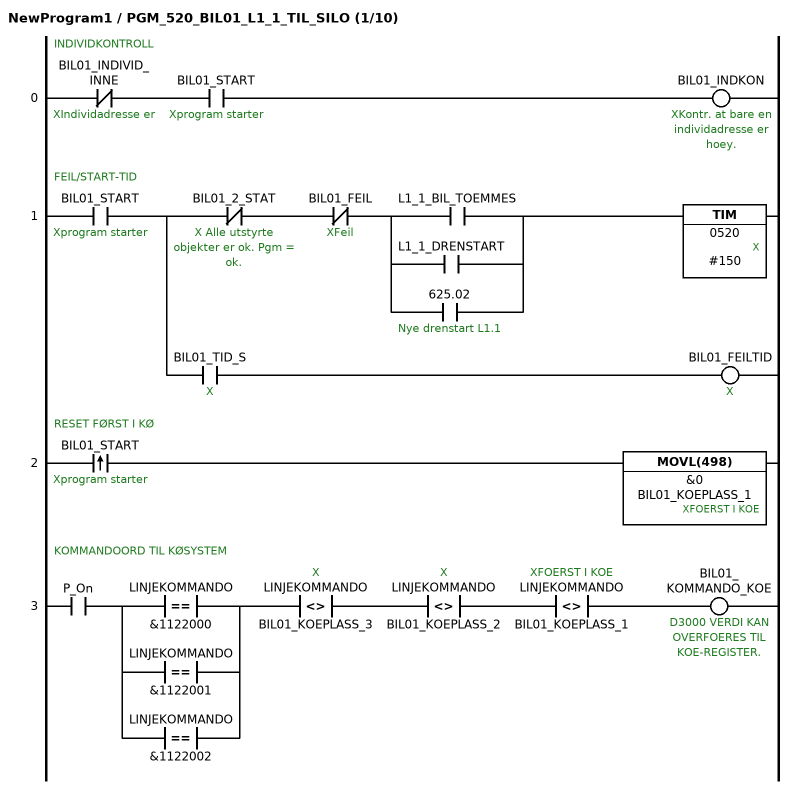
; [picture p576: NewProgram1 / PGM_520_BIL01_L1_1_TIL_SILO, rungs 0-3]
; rung 0: INDIVIDKONTROLL
LDNOT BIL01_INDIVID_INNE  ; XIndividadresse er
AND BIL01_START  ; Xprogram starter
OUT BIL01_INDKON  ; XKontr. at bare en individadresse er hoey.
; rung 1: FEIL/START-TID
LD BIL01_START  ; Xprogram starter
OUT TR0
ANDNOT BIL01_2_STAT  ; X Alle utstyrte objekter er ok. Pgm = ok.
ANDNOT BIL01_FEIL  ; XFeil
LD L1_1_BIL_TOEMMES
OR L1_1_DRENSTART
OR 625.02  ; Nye drenstart L1.1
ANDLD
TIM 0520 #150  ; X
LD TR0
AND BIL01_TID_S  ; X
OUT BIL01_FEILTID  ; X
; rung 2: RESET FØRST I KØ
@LD BIL01_START  ; Xprogram starter
MOVL(498) &0 BIL01_KOEPLASS_1  ; XFOERST I KOE
; rung 3: KOMMANDOORD TIL KØSYSTEM
LD P_On
LD=L(301) LINJEKOMMANDO &1122000
OR=L(301) LINJEKOMMANDO &1122001
OR=L(301) LINJEKOMMANDO &1122002
ANDLD
AND<>L(306) LINJEKOMMANDO BIL01_KOEPLASS_3  ; X
AND<>L(306) LINJEKOMMANDO BIL01_KOEPLASS_2  ; X
AND<>L(306) LINJEKOMMANDO BIL01_KOEPLASS_1  ; XFOERST I KOE
OUT BIL01_KOMMANDO_KOE  ; D3000 VERDI KAN OVERFOERES TIL KOE-REGISTER.

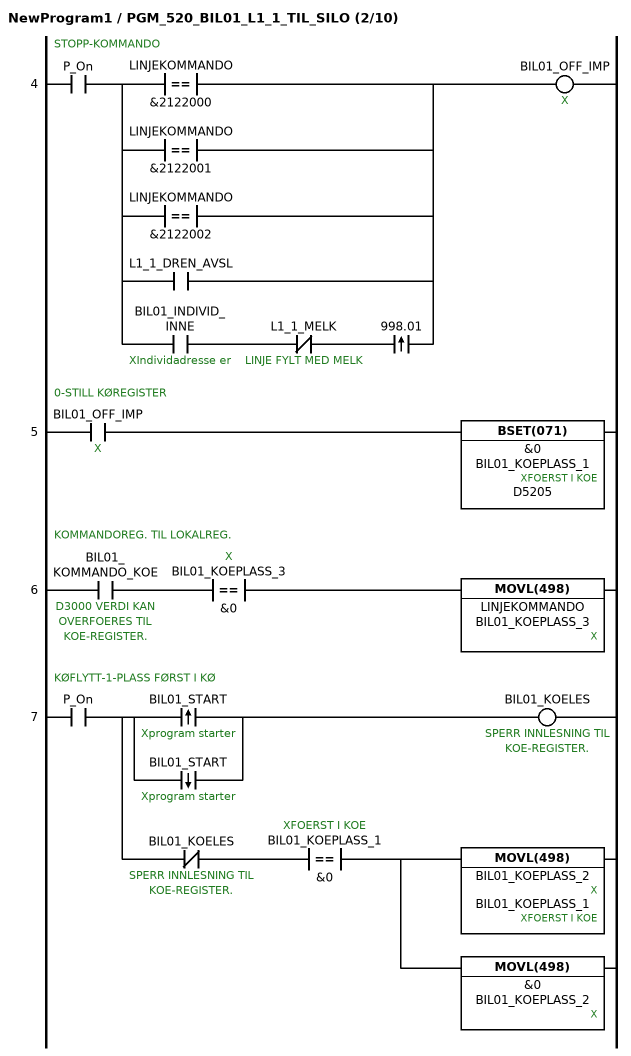
; rung 4: STOPP-KOMMANDO
LD P_On
LD=L(301) LINJEKOMMANDO &2122000
OR=L(301) LINJEKOMMANDO &2122001
OR=L(301) LINJEKOMMANDO &2122002
OR L1_1_DREN_AVSL
LD BIL01_INDIVID_INNE  ; XIndividadresse er
ANDNOT L1_1_MELK  ; LINJE FYLT MED MELK
@AND 998.01
ORLD
ANDLD
OUT BIL01_OFF_IMP  ; X
; rung 5: 0-STILL KØREGISTER
LD BIL01_OFF_IMP  ; X
BSET(071) &0 BIL01_KOEPLASS_1 D5205  ; XFOERST I KOE
; rung 6: KOMMANDOREG. TIL LOKALREG.
LD BIL01_KOMMANDO_KOE  ; D3000 VERDI KAN OVERFOERES TIL KOE-REGISTER.
AND=L(301) BIL01_KOEPLASS_3 &0  ; X
MOVL(498) LINJEKOMMANDO BIL01_KOEPLASS_3  ; X
; rung 7: KØFLYTT-1-PLASS FØRST I KØ
LD P_On
OUT TR0
@LD BIL01_START  ; Xprogram starter
%OR BIL01_START  ; Xprogram starter
ANDLD
OUT BIL01_KOELES  ; SPERR INNLESNING TIL KOE-REGISTER.
LD TR0
ANDNOT BIL01_KOELES  ; SPERR INNLESNING TIL KOE-REGISTER.
AND=L(301) BIL01_KOEPLASS_1 &0  ; XFOERST I KOE
MOVL(498) BIL01_KOEPLASS_2 BIL01_KOEPLASS_1  ; X, XFOERST I KOE
MOVL(498) &0 BIL01_KOEPLASS_2  ; X

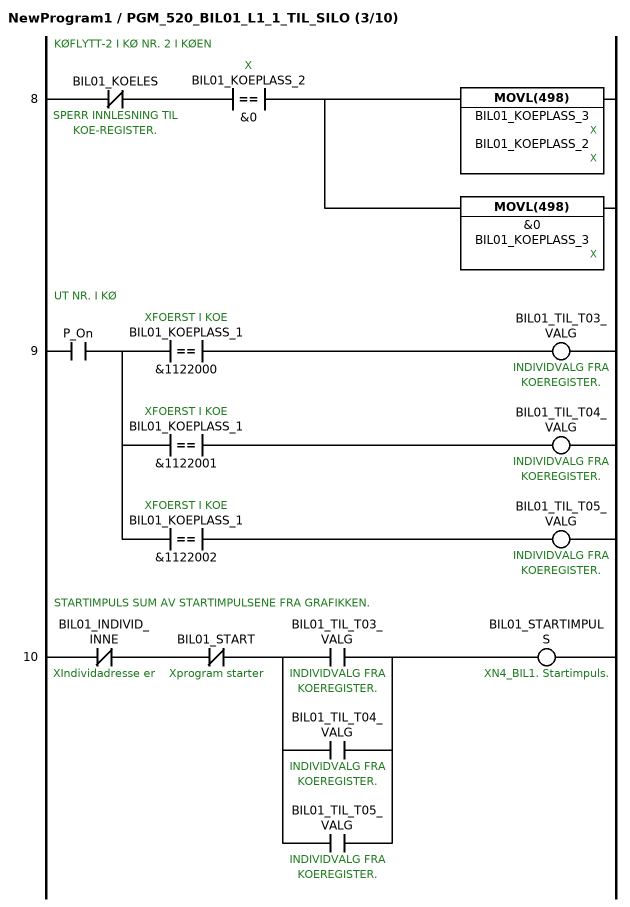
; rung 8: KØFLYTT-2 I KØ NR. 2 I KØEN
LDNOT BIL01_KOELES  ; SPERR INNLESNING TIL KOE-REGISTER.
AND=L(301) BIL01_KOEPLASS_2 &0  ; X
MOVL(498) BIL01_KOEPLASS_3 BIL01_KOEPLASS_2  ; X
MOVL(498) &0 BIL01_KOEPLASS_3  ; X
; rung 9: UT NR. I KØ
LD P_On
OUT TR0
AND=L(301) BIL01_KOEPLASS_1 &1122000  ; XFOERST I KOE
OUT BIL01_TIL_T03_VALG  ; INDIVIDVALG FRA KOEREGISTER.
LD TR0
AND=L(301) BIL01_KOEPLASS_1 &1122001  ; XFOERST I KOE
OUT BIL01_TIL_T04_VALG  ; INDIVIDVALG FRA KOEREGISTER.
LD TR0
AND=L(301) BIL01_KOEPLASS_1 &1122002  ; XFOERST I KOE
OUT BIL01_TIL_T05_VALG  ; INDIVIDVALG FRA KOEREGISTER.
; rung 10: STARTIMPULS SUM AV STARTIMPULSENE FRA GRAFIKKEN.
LDNOT BIL01_INDIVID_INNE  ; XIndividadresse er
ANDNOT BIL01_START  ; Xprogram starter
LD BIL01_TIL_T03_VALG  ; INDIVIDVALG FRA KOEREGISTER.
OR BIL01_TIL_T04_VALG  ; INDIVIDVALG FRA KOEREGISTER.
OR BIL01_TIL_T05_VALG  ; INDIVIDVALG FRA KOEREGISTER.
ANDLD
OUT BIL01_STARTIMPULS  ; XN4_BIL1. Startimpuls.

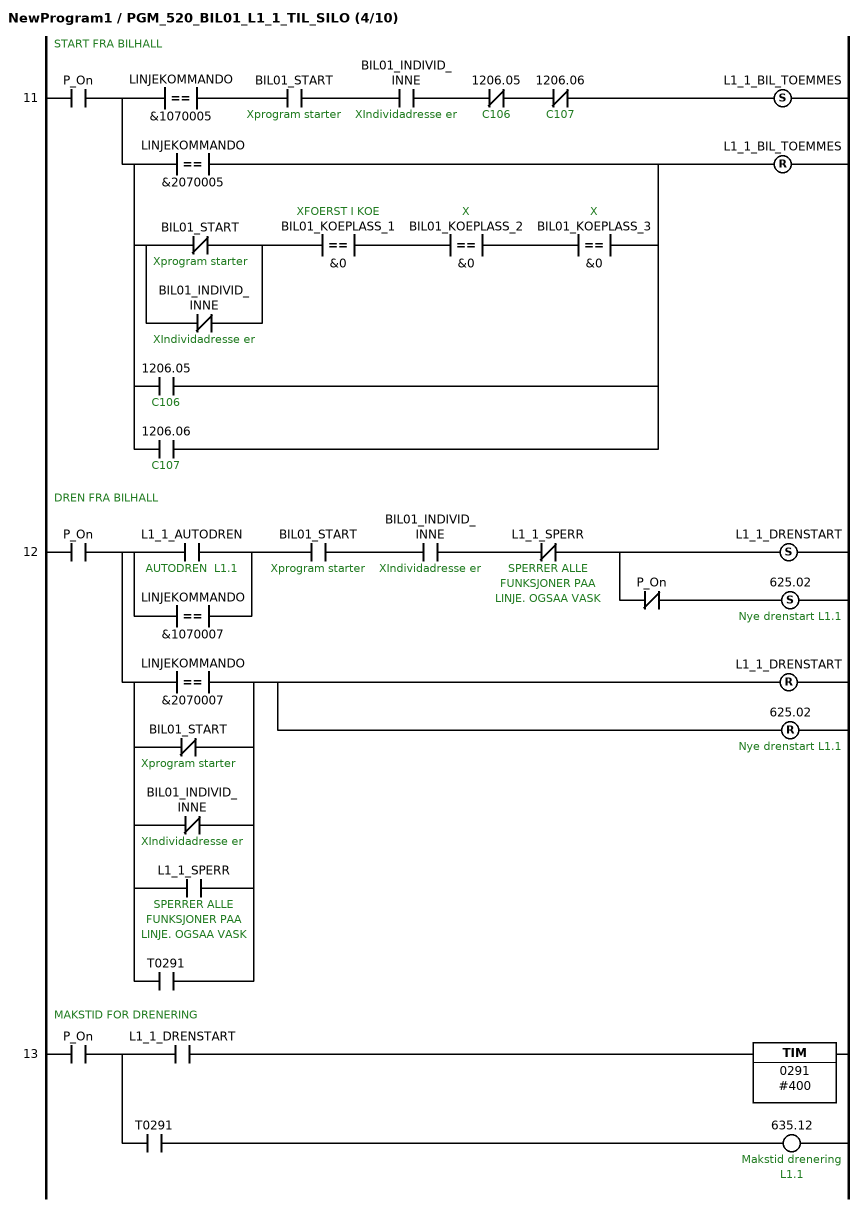
; rung 11: START FRA BILHALL
LD P_On
OUT TR0
AND=L(301) LINJEKOMMANDO &1070005
AND BIL01_START  ; Xprogram starter
AND BIL01_INDIVID_INNE  ; XIndividadresse er
ANDNOT 1206.05  ; C106
ANDNOT 1206.06  ; C107
SET L1_1_BIL_TOEMMES
LD TR0
LD=L(301) LINJEKOMMANDO &2070005
LDNOT BIL01_START  ; Xprogram starter
ORNOT BIL01_INDIVID_INNE  ; XIndividadresse er
AND=(300) BIL01_KOEPLASS_1 &0  ; XFOERST I KOE
AND=(300) BIL01_KOEPLASS_2 &0  ; X
AND=(300) BIL01_KOEPLASS_3 &0  ; X
ORLD
OR 1206.05  ; C106
OR 1206.06  ; C107
ANDLD
RSET L1_1_BIL_TOEMMES
; rung 12: DREN FRA BILHALL
LD P_On
OUT TR0
LD L1_1_AUTODREN  ; AUTODREN  L1.1
OR=L(301) LINJEKOMMANDO &1070007
ANDLD
AND BIL01_START  ; Xprogram starter
AND BIL01_INDIVID_INNE  ; XIndividadresse er
ANDNOT L1_1_SPERR  ; SPERRER ALLE FUNKSJONER PAA LINJE. OGSAA VASK
SET L1_1_DRENSTART
ANDNOT P_On
SET 625.02  ; Nye drenstart L1.1
LD TR0
LD=L(301) LINJEKOMMANDO &2070007
ORNOT BIL01_START  ; Xprogram starter
ORNOT BIL01_INDIVID_INNE  ; XIndividadresse er
OR L1_1_SPERR  ; SPERRER ALLE FUNKSJONER PAA LINJE. OGSAA VASK
OR T0291
ANDLD
RSET L1_1_DRENSTART
RSET 625.02  ; Nye drenstart L1.1
; rung 13: MAKSTID FOR DRENERING
LD P_On
OUT TR0
AND L1_1_DRENSTART
TIM 0291 #400
LD TR0
AND T0291
OUT 635.12  ; Makstid drenering L1.1

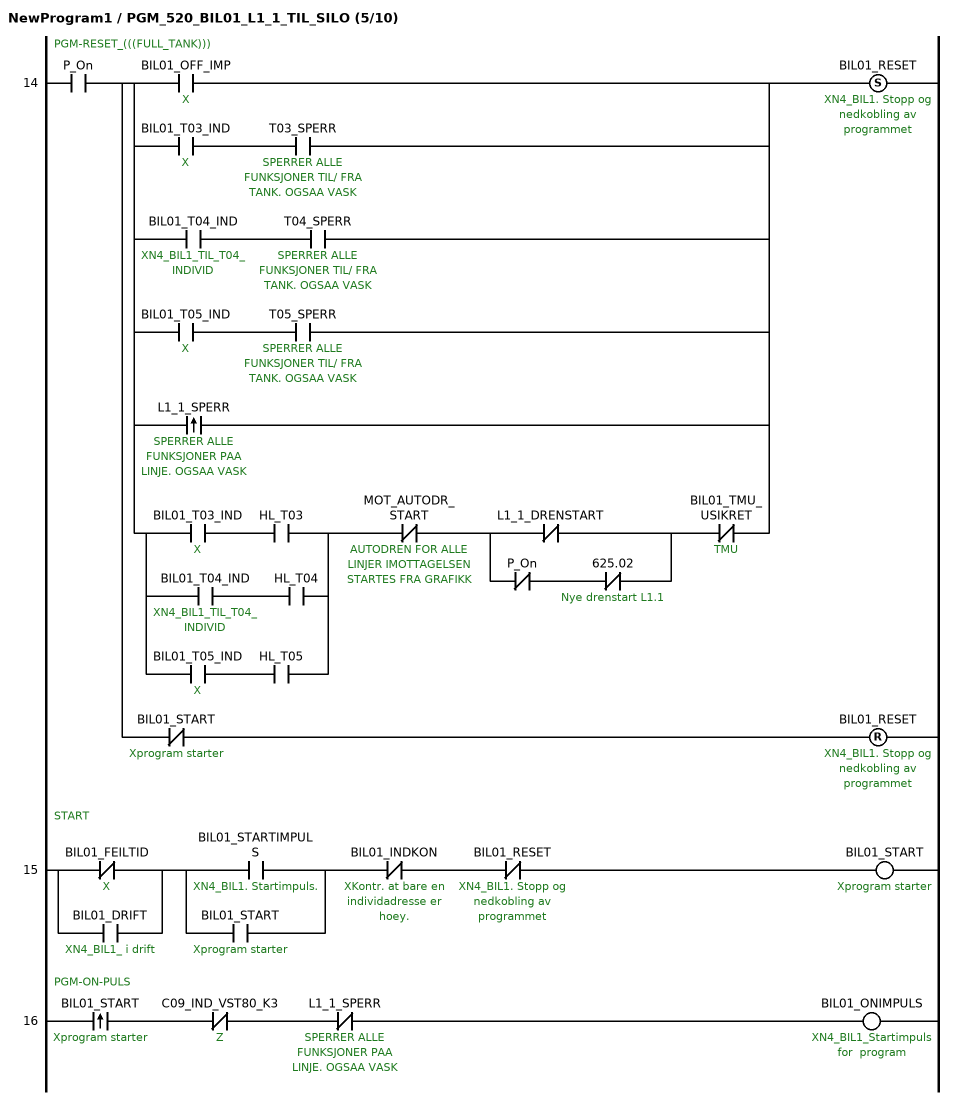
; rung 14: PGM-RESET_(((FULL_TANK)))
LD P_On
OUT TR0
LD BIL01_OFF_IMP  ; X
LD BIL01_T03_IND  ; X
AND T03_SPERR  ; SPERRER ALLE FUNKSJONER TIL/ FRA TANK. OGSAA VASK
ORLD
LD BIL01_T04_IND  ; XN4_BIL1_TIL_T04_INDIVID
AND T04_SPERR  ; SPERRER ALLE FUNKSJONER TIL/ FRA TANK. OGSAA VASK
ORLD
LD BIL01_T05_IND  ; X
AND T05_SPERR  ; SPERRER ALLE FUNKSJONER TIL/ FRA TANK. OGSAA VASK
ORLD
@OR L1_1_SPERR  ; SPERRER ALLE FUNKSJONER PAA LINJE. OGSAA VASK
LD BIL01_T03_IND  ; X
AND HL_T03
LD BIL01_T04_IND  ; XN4_BIL1_TIL_T04_INDIVID
AND HL_T04
ORLD
LD BIL01_T05_IND  ; X
AND HL_T05
ORLD
ANDNOT MOT_AUTODR_START  ; AUTODREN FOR ALLE LINJER IMOTTAGELSEN STARTES FRA GRAFIKK
LDNOT L1_1_DRENSTART
LDNOT P_On
ANDNOT 625.02  ; Nye drenstart L1.1
ORLD
ANDLD
ANDNOT BIL01_TMU_USIKRET  ; TMU
ORLD
ANDLD
SET BIL01_RESET  ; XN4_BIL1. Stopp og nedkobling av programmet
LD TR0
ANDNOT BIL01_START  ; Xprogram starter
RSET BIL01_RESET  ; XN4_BIL1. Stopp og nedkobling av programmet
; rung 15: START
LDNOT BIL01_FEILTID  ; X
OR BIL01_DRIFT  ; XN4_BIL1_ i drift
LD BIL01_STARTIMPULS  ; XN4_BIL1. Startimpuls.
OR BIL01_START  ; Xprogram starter
ANDLD
ANDNOT BIL01_INDKON  ; XKontr. at bare en individadresse er hoey.
ANDNOT BIL01_RESET  ; XN4_BIL1. Stopp og nedkobling av programmet
OUT BIL01_START  ; Xprogram starter
; rung 16: PGM-ON-PULS
@LD BIL01_START  ; Xprogram starter
ANDNOT C09_IND_VST80_K3  ; Z
ANDNOT L1_1_SPERR  ; SPERRER ALLE FUNKSJONER PAA LINJE. OGSAA VASK
OUT BIL01_ONIMPULS  ; XN4_BIL1_Startimpuls for  program

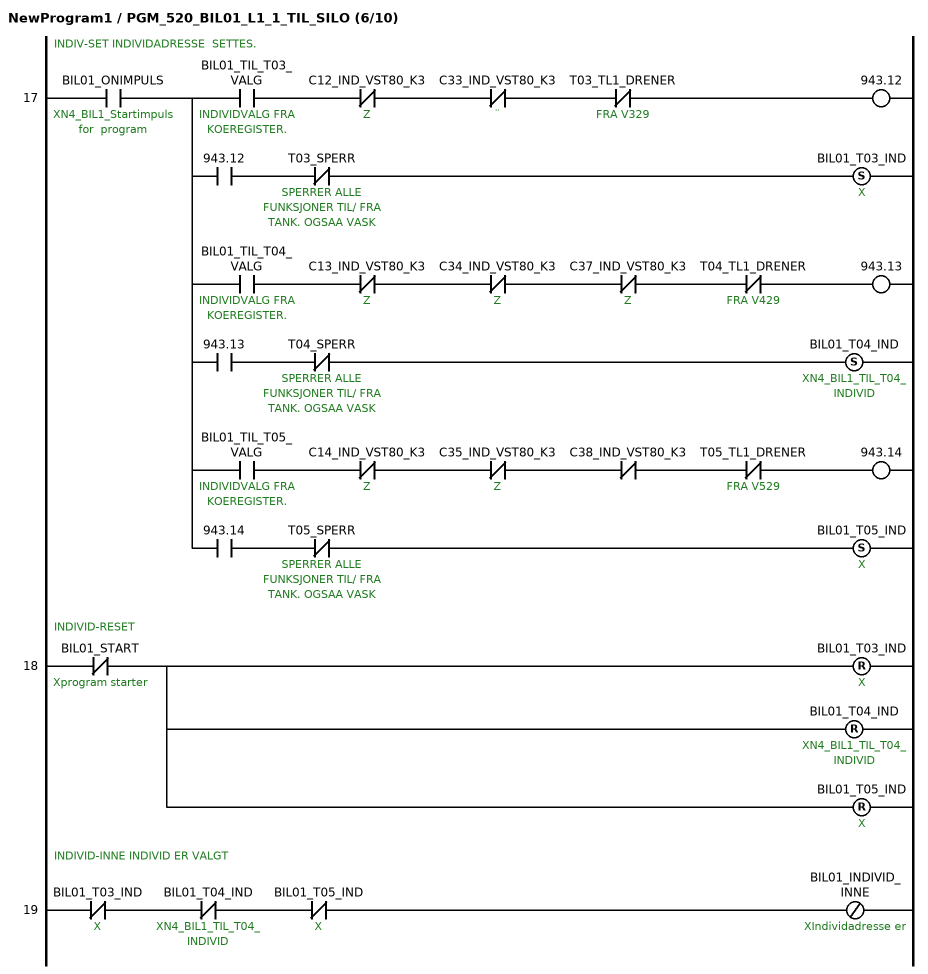
; rung 17: INDIV-SET INDIVIDADRESSE  SETTES.
LD BIL01_ONIMPULS  ; XN4_BIL1_Startimpuls for  program
OUT TR0
AND BIL01_TIL_T03_VALG  ; INDIVIDVALG FRA KOEREGISTER.
ANDNOT C12_IND_VST80_K3  ; Z
ANDNOT C33_IND_VST80_K3  ; ¨
ANDNOT T03_TL1_DRENER  ; FRA V329
OUT 943.12
LD TR0
AND 943.12
ANDNOT T03_SPERR  ; SPERRER ALLE FUNKSJONER TIL/ FRA TANK. OGSAA VASK
SET BIL01_T03_IND  ; X
LD TR0
AND BIL01_TIL_T04_VALG  ; INDIVIDVALG FRA KOEREGISTER.
ANDNOT C13_IND_VST80_K3  ; Z
ANDNOT C34_IND_VST80_K3  ; Z
ANDNOT C37_IND_VST80_K3  ; Z
ANDNOT T04_TL1_DRENER  ; FRA V429
OUT 943.13
LD TR0
AND 943.13
ANDNOT T04_SPERR  ; SPERRER ALLE FUNKSJONER TIL/ FRA TANK. OGSAA VASK
SET BIL01_T04_IND  ; XN4_BIL1_TIL_T04_INDIVID
LD TR0
AND BIL01_TIL_T05_VALG  ; INDIVIDVALG FRA KOEREGISTER.
ANDNOT C14_IND_VST80_K3  ; Z
ANDNOT C35_IND_VST80_K3  ; Z
ANDNOT C38_IND_VST80_K3
ANDNOT T05_TL1_DRENER  ; FRA V529
OUT 943.14
LD TR0
AND 943.14
ANDNOT T05_SPERR  ; SPERRER ALLE FUNKSJONER TIL/ FRA TANK. OGSAA VASK
SET BIL01_T05_IND  ; X
; rung 18: INDIVID-RESET
LDNOT BIL01_START  ; Xprogram starter
RSET BIL01_T03_IND  ; X
RSET BIL01_T04_IND  ; XN4_BIL1_TIL_T04_INDIVID
RSET BIL01_T05_IND  ; X
; rung 19: INDIVID-INNE INDIVID ER VALGT
LDNOT BIL01_T03_IND  ; X
ANDNOT BIL01_T04_IND  ; XN4_BIL1_TIL_T04_INDIVID
ANDNOT BIL01_T05_IND  ; X
OUTNOT BIL01_INDIVID_INNE  ; XIndividadresse er

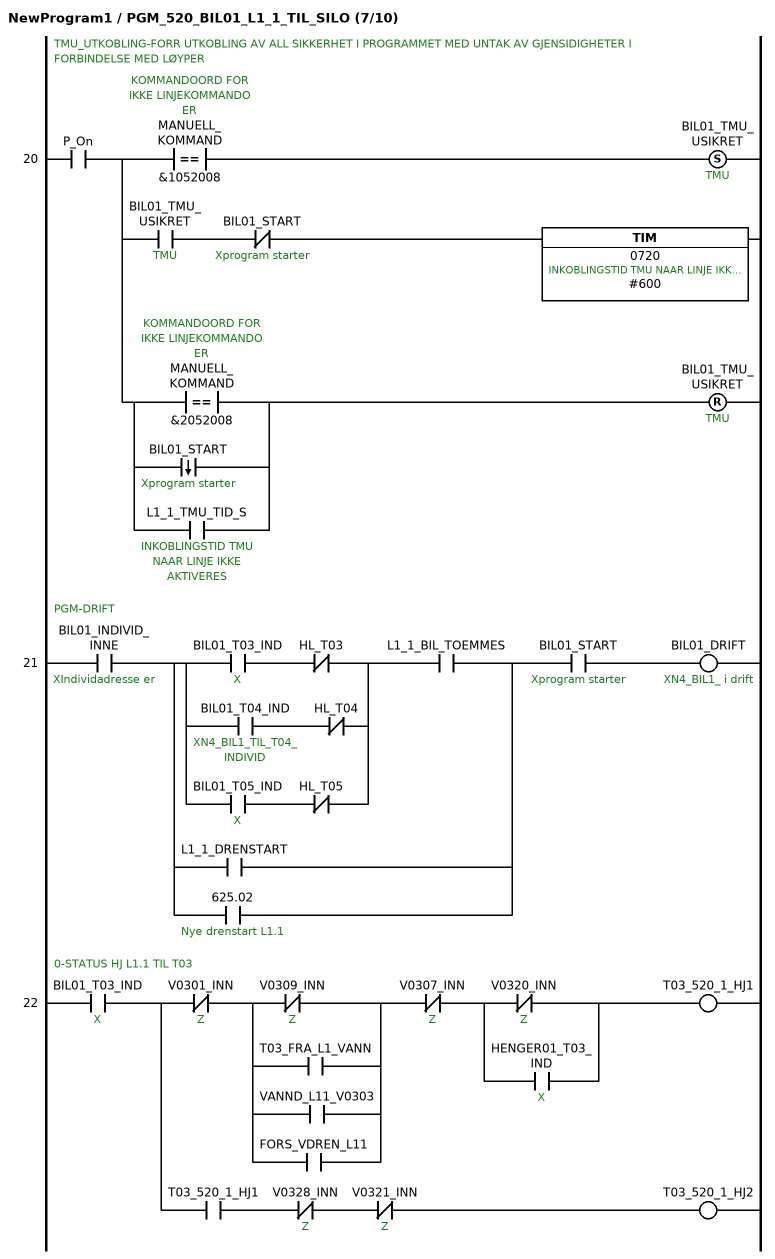
; rung 20: TMU_UTKOBLING-FORR UTKOBLING AV ALL SIKKERHET I PROGRAMMET MED UNTAK AV GJENSIDIGHETER I FORBINDELSE MED LØYPER
LD P_On
OUT TR0
AND=L(301) MANUELL_KOMMAND &1052008  ; KOMMANDOORD FOR IKKE LINJEKOMMANDOER
SET BIL01_TMU_USIKRET  ; TMU
LD TR0
AND BIL01_TMU_USIKRET  ; TMU
ANDNOT BIL01_START  ; Xprogram starter
TIM 0720 #600  ; INKOBLINGSTID TMU NAAR LINJE IKKE AKTIVERES
LD TR0
LD=L(301) MANUELL_KOMMAND &2052008  ; KOMMANDOORD FOR IKKE LINJEKOMMANDOER
%OR BIL01_START  ; Xprogram starter
OR L1_1_TMU_TID_S  ; INKOBLINGSTID TMU NAAR LINJE IKKE AKTIVERES
ANDLD
RSET BIL01_TMU_USIKRET  ; TMU
; rung 21: PGM-DRIFT
LD BIL01_INDIVID_INNE  ; XIndividadresse er
LD BIL01_T03_IND  ; X
ANDNOT HL_T03
LD BIL01_T04_IND  ; XN4_BIL1_TIL_T04_INDIVID
ANDNOT HL_T04
ORLD
LD BIL01_T05_IND  ; X
ANDNOT HL_T05
ORLD
AND L1_1_BIL_TOEMMES
OR L1_1_DRENSTART
OR 625.02  ; Nye drenstart L1.1
ANDLD
AND BIL01_START  ; Xprogram starter
OUT BIL01_DRIFT  ; XN4_BIL1_ i drift
; rung 22: 0-STATUS HJ L1.1 TIL T03
LD BIL01_T03_IND  ; X
OUT TR0
ANDNOT V0301_INN  ; Z
LDNOT V0309_INN  ; Z
OR T03_FRA_L1_VANN
OR VANND_L11_V0303
OR FORS_VDREN_L11
ANDLD
ANDNOT V0307_INN  ; Z
LDNOT V0320_INN  ; Z
OR HENGER01_T03_IND  ; X
ANDLD
OUT T03_520_1_HJ1
LD TR0
AND T03_520_1_HJ1
ANDNOT V0328_INN  ; Z
ANDNOT V0321_INN  ; Z
OUT T03_520_1_HJ2

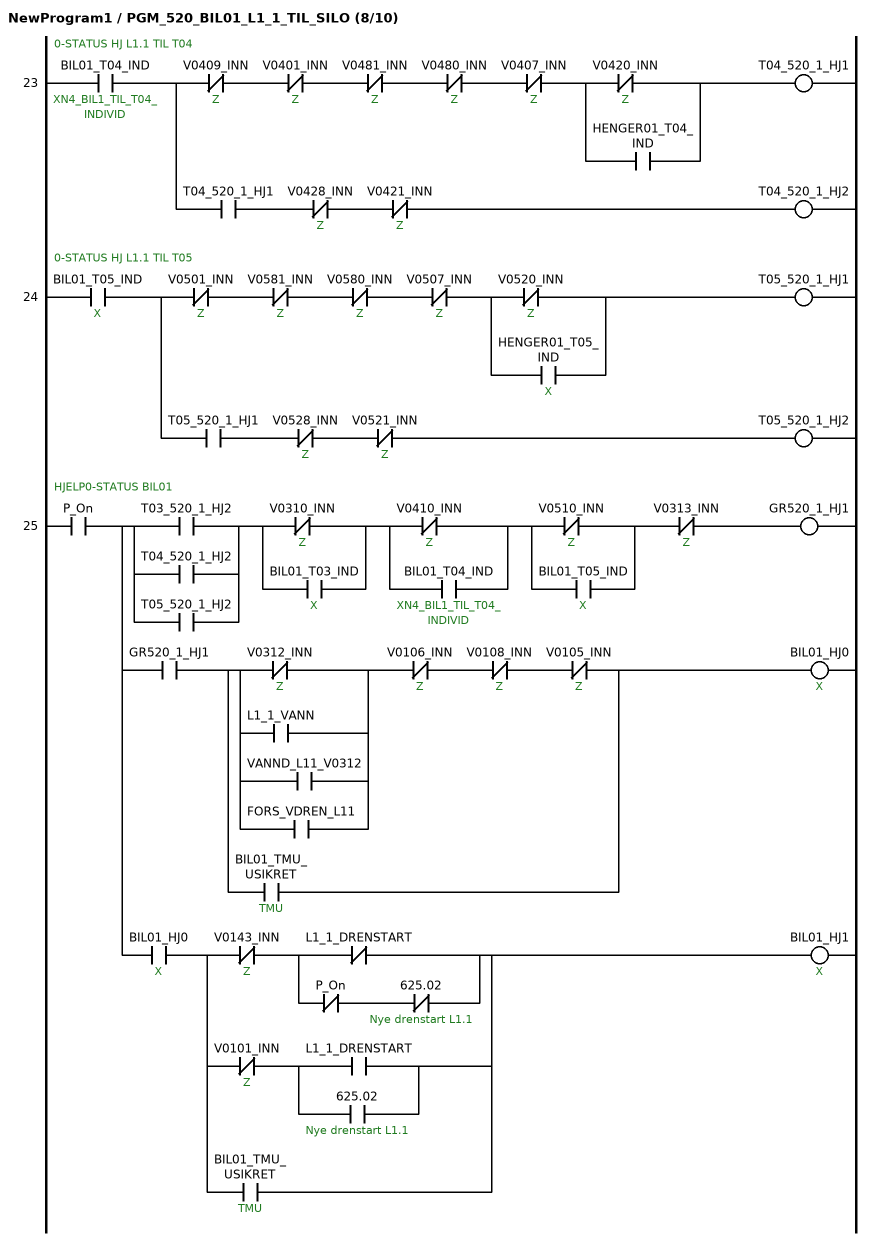
; rung 23: 0-STATUS HJ L1.1 TIL T04
LD BIL01_T04_IND  ; XN4_BIL1_TIL_T04_INDIVID
OUT TR0
ANDNOT V0409_INN  ; Z
ANDNOT V0401_INN  ; Z
ANDNOT V0481_INN  ; Z
ANDNOT V0480_INN  ; Z
ANDNOT V0407_INN  ; Z
LDNOT V0420_INN  ; Z
OR HENGER01_T04_IND
ANDLD
OUT T04_520_1_HJ1
LD TR0
AND T04_520_1_HJ1
ANDNOT V0428_INN  ; Z
ANDNOT V0421_INN  ; Z
OUT T04_520_1_HJ2
; rung 24: 0-STATUS HJ L1.1 TIL T05
LD BIL01_T05_IND  ; X
OUT TR0
ANDNOT V0501_INN  ; Z
ANDNOT V0581_INN  ; Z
ANDNOT V0580_INN  ; Z
ANDNOT V0507_INN  ; Z
LDNOT V0520_INN  ; Z
OR HENGER01_T05_IND  ; X
ANDLD
OUT T05_520_1_HJ1
LD TR0
AND T05_520_1_HJ1
ANDNOT V0528_INN  ; Z
ANDNOT V0521_INN  ; Z
OUT T05_520_1_HJ2
; rung 25: HJELP0-STATUS BIL01
LD P_On
OUT TR0
LD T03_520_1_HJ2
OR T04_520_1_HJ2
OR T05_520_1_HJ2
ANDLD
LDNOT V0310_INN  ; Z
OR BIL01_T03_IND  ; X
ANDLD
LDNOT V0410_INN  ; Z
OR BIL01_T04_IND  ; XN4_BIL1_TIL_T04_INDIVID
ANDLD
LDNOT V0510_INN  ; Z
OR BIL01_T05_IND  ; X
ANDLD
ANDNOT V0313_INN  ; Z
OUT GR520_1_HJ1
LD TR0
AND GR520_1_HJ1
LDNOT V0312_INN  ; Z
OR L1_1_VANN
OR VANND_L11_V0312
OR FORS_VDREN_L11
ANDNOT V0106_INN  ; Z
ANDNOT V0108_INN  ; Z
ANDNOT V0105_INN  ; Z
OR BIL01_TMU_USIKRET  ; TMU
ANDLD
OUT BIL01_HJ0  ; X
LD TR0
AND BIL01_HJ0  ; X
LDNOT V0143_INN  ; Z
LDNOT L1_1_DRENSTART
LDNOT P_On
ANDNOT 625.02  ; Nye drenstart L1.1
ORLD
ANDLD
LDNOT V0101_INN  ; Z
LD L1_1_DRENSTART
OR 625.02  ; Nye drenstart L1.1
ANDLD
ORLD
OR BIL01_TMU_USIKRET  ; TMU
ANDLD
OUT BIL01_HJ1  ; X

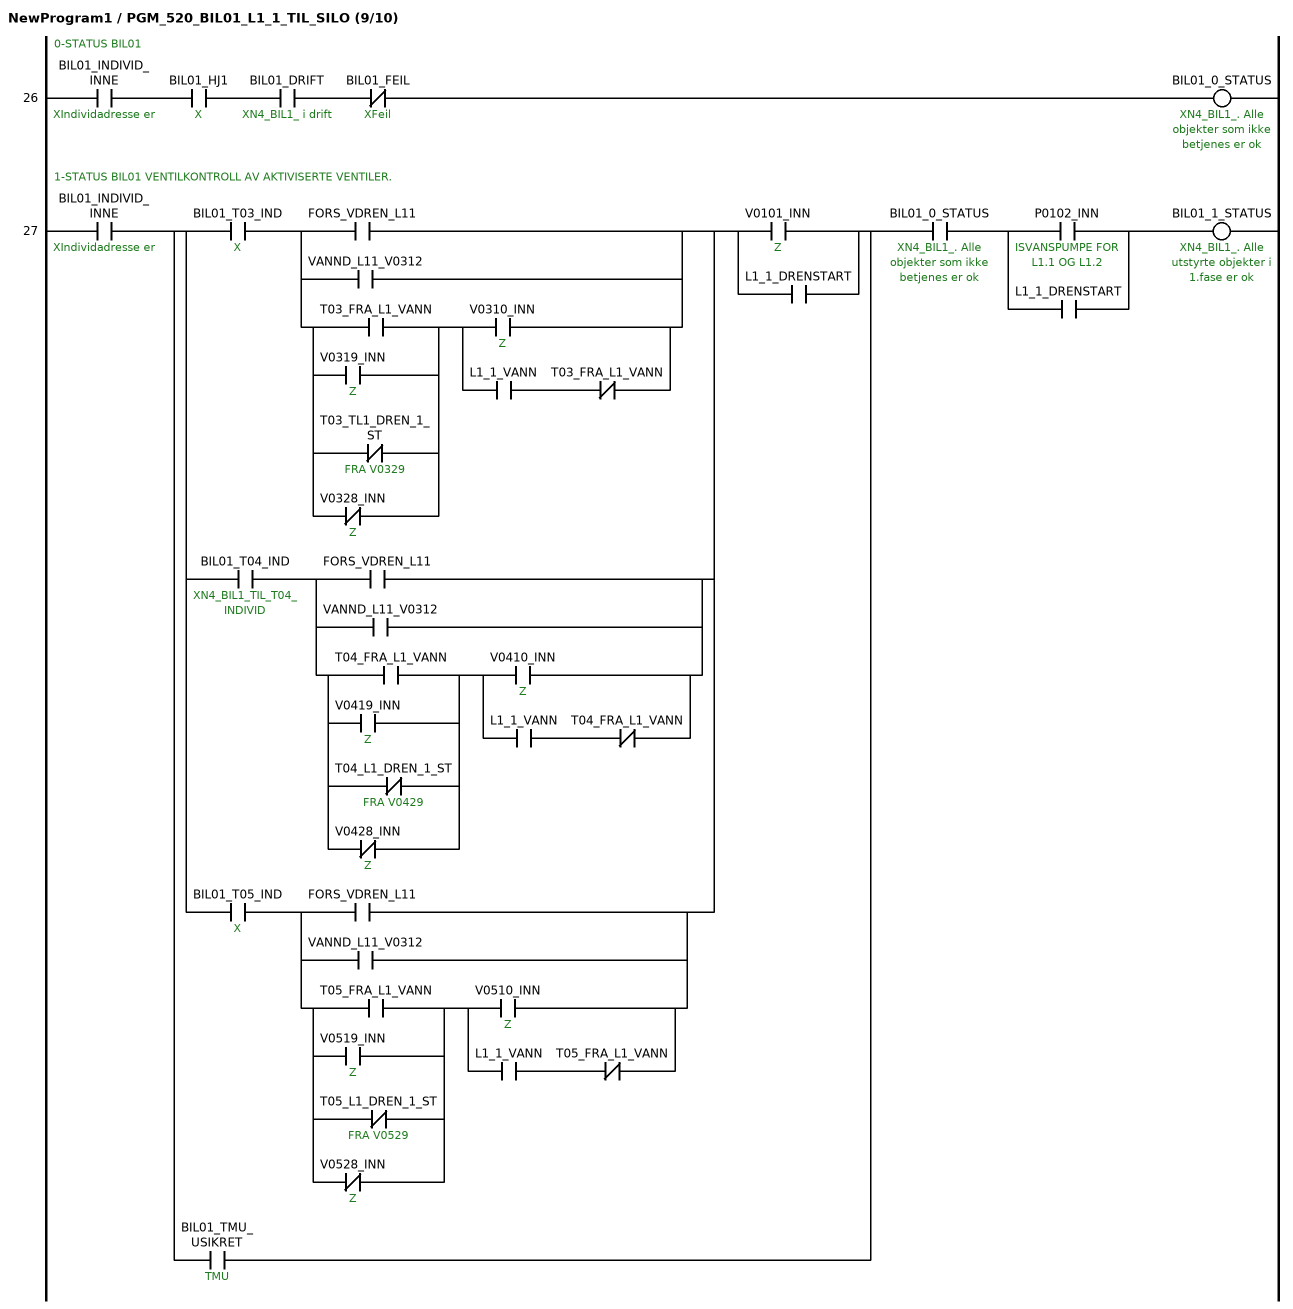
; rung 26: 0-STATUS BIL01
LD BIL01_INDIVID_INNE  ; XIndividadresse er
AND BIL01_HJ1  ; X
AND BIL01_DRIFT  ; XN4_BIL1_ i drift
ANDNOT BIL01_FEIL  ; XFeil
OUT BIL01_0_STATUS  ; XN4_BIL1_. Alle objekter som ikke betjenes er ok
; rung 27: 1-STATUS BIL01 VENTILKONTROLL AV AKTIVISERTE VENTILER.
LD BIL01_INDIVID_INNE  ; XIndividadresse er
LD BIL01_T03_IND  ; X
LD FORS_VDREN_L11
OR VANND_L11_V0312
LD T03_FRA_L1_VANN
OR V0319_INN  ; Z
ORNOT T03_TL1_DREN_1_ST  ; FRA V0329
ORNOT V0328_INN  ; Z
LD V0310_INN  ; Z
LD L1_1_VANN
ANDNOT T03_FRA_L1_VANN
ORLD
ANDLD
ORLD
ANDLD
LD BIL01_T04_IND  ; XN4_BIL1_TIL_T04_INDIVID
LD FORS_VDREN_L11
OR VANND_L11_V0312
LD T04_FRA_L1_VANN
OR V0419_INN  ; Z
ORNOT T04_L1_DREN_1_ST  ; FRA V0429
ORNOT V0428_INN  ; Z
LD V0410_INN  ; Z
LD L1_1_VANN
ANDNOT T04_FRA_L1_VANN
ORLD
ANDLD
ORLD
ANDLD
ORLD
LD BIL01_T05_IND  ; X
LD FORS_VDREN_L11
OR VANND_L11_V0312
LD T05_FRA_L1_VANN
OR V0519_INN  ; Z
ORNOT T05_L1_DREN_1_ST  ; FRA V0529
ORNOT V0528_INN  ; Z
LD V0510_INN  ; Z
LD L1_1_VANN
ANDNOT T05_FRA_L1_VANN
ORLD
ANDLD
ORLD
ANDLD
ORLD
LD V0101_INN  ; Z
OR L1_1_DRENSTART
ANDLD
OR BIL01_TMU_USIKRET  ; TMU
ANDLD
AND BIL01_0_STATUS  ; XN4_BIL1_. Alle objekter som ikke betjenes er ok
LD P0102_INN  ; ISVANSPUMPE FOR L1.1 OG L1.2
OR L1_1_DRENSTART
ANDLD
OUT BIL01_1_STATUS  ; XN4_BIL1_. Alle utstyrte objekter i 1.fase er ok

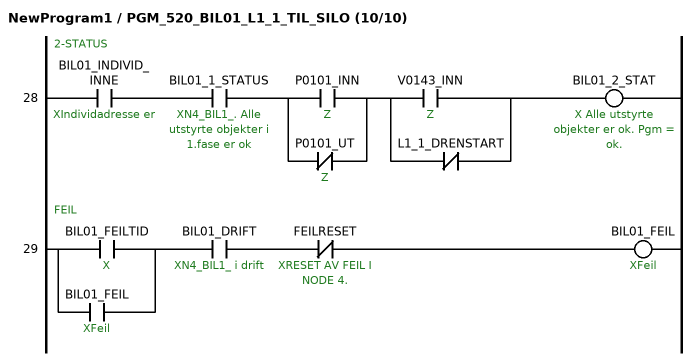
; rung 28: 2-STATUS
LD BIL01_INDIVID_INNE  ; XIndividadresse er
AND BIL01_1_STATUS  ; XN4_BIL1_. Alle utstyrte objekter i 1.fase er ok
LD P0101_INN  ; Z
ORNOT P0101_UT  ; Z
ANDLD
LD V0143_INN  ; Z
ORNOT L1_1_DRENSTART
ANDLD
OUT BIL01_2_STAT  ; X Alle utstyrte objekter er ok. Pgm = ok.
; rung 29: FEIL
LD BIL01_FEILTID  ; X
OR BIL01_FEIL  ; XFeil
AND BIL01_DRIFT  ; XN4_BIL1_ i drift
ANDNOT FEILRESET  ; XRESET AV FEIL I NODE 4.
OUT BIL01_FEIL  ; XFeil
; rung 30: Ingen_kommentar_funnet

### Section V0104_P0101

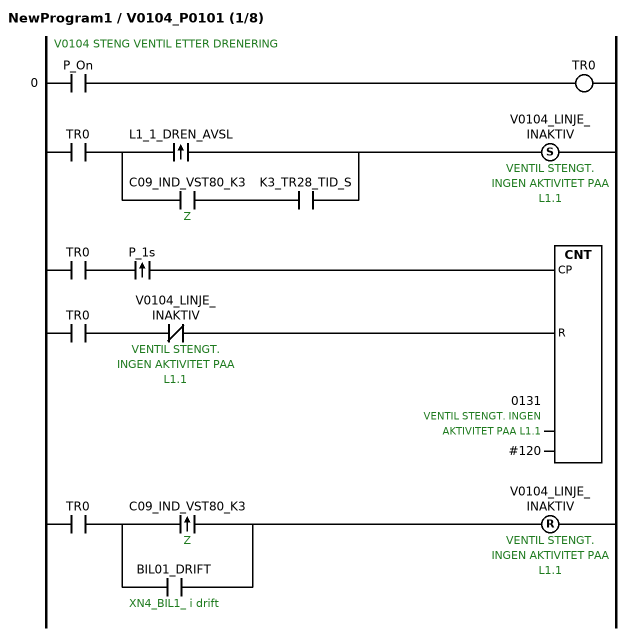
; rung 0: V0104 STENG VENTIL ETTER DRENERING
LD P_On
OUT TR0
@LD L1_1_DREN_AVSL
LD C09_IND_VST80_K3  ; Z
AND K3_TR28_TID_S
ORLD
ANDLD
SET V0104_LINJE_INAKTIV  ; VENTIL STENGT. INGEN AKTIVITET PAA L1.1
LD TR0
@AND P_1s
LD TR0
ANDNOT V0104_LINJE_INAKTIV  ; VENTIL STENGT. INGEN AKTIVITET PAA L1.1
CNT 0131 #120  ; VENTIL STENGT. INGEN AKTIVITET PAA L1.1
LD TR0
@LD C09_IND_VST80_K3  ; Z
OR BIL01_DRIFT  ; XN4_BIL1_ i drift
ANDLD
RSET V0104_LINJE_INAKTIV  ; VENTIL STENGT. INGEN AKTIVITET PAA L1.1

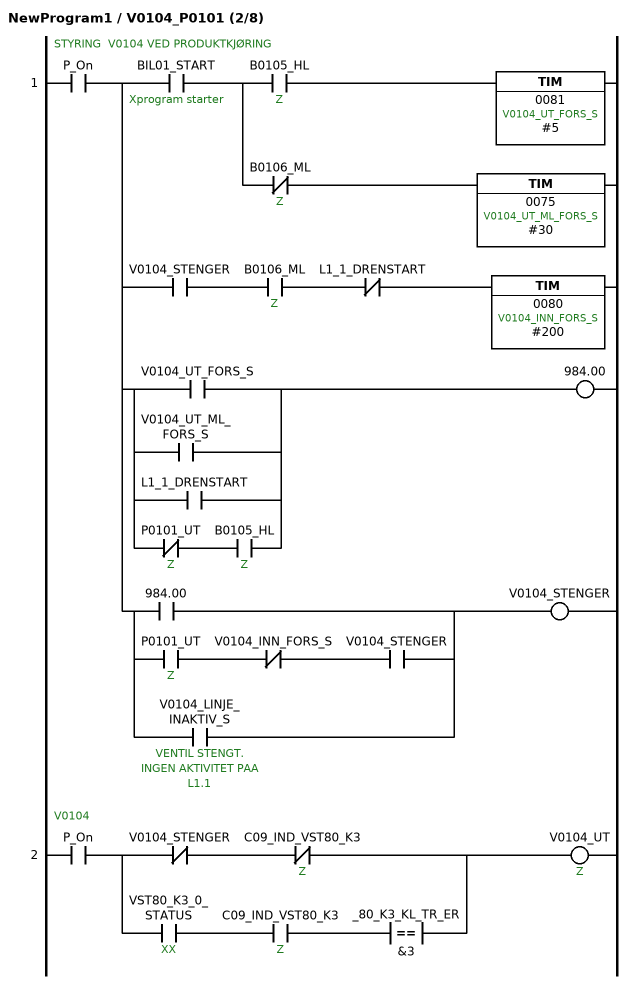
; rung 1: STYRING  V0104 VED PRODUKTKJØRING
LD P_On
OUT TR0
AND BIL01_START  ; Xprogram starter
OUT TR1
AND B0105_HL  ; Z
TIM 0081 #5  ; V0104_UT_FORS_S
LD TR1
ANDNOT B0106_ML  ; Z
TIM 0075 #30  ; V0104_UT_ML_FORS_S
LD TR0
AND V0104_STENGER
AND B0106_ML  ; Z
ANDNOT L1_1_DRENSTART
TIM 0080 #200  ; V0104_INN_FORS_S
LD TR0
LD V0104_UT_FORS_S
OR V0104_UT_ML_FORS_S
OR L1_1_DRENSTART
LDNOT P0101_UT  ; Z
AND B0105_HL  ; Z
ORLD
ANDLD
OUT 984.00
LD TR0
LD 984.00
LD P0101_UT  ; Z
ANDNOT V0104_INN_FORS_S
AND V0104_STENGER
ORLD
OR V0104_LINJE_INAKTIV_S  ; VENTIL STENGT. INGEN AKTIVITET PAA L1.1
ANDLD
OUT V0104_STENGER
; rung 2: V0104
LD P_On
LDNOT V0104_STENGER
ANDNOT C09_IND_VST80_K3  ; Z
LD VST80_K3_0_STATUS  ; XX
AND C09_IND_VST80_K3  ; Z
AND=(300) _80_K3_KL_TR_ER &3
ORLD
ANDLD
OUT V0104_UT  ; Z

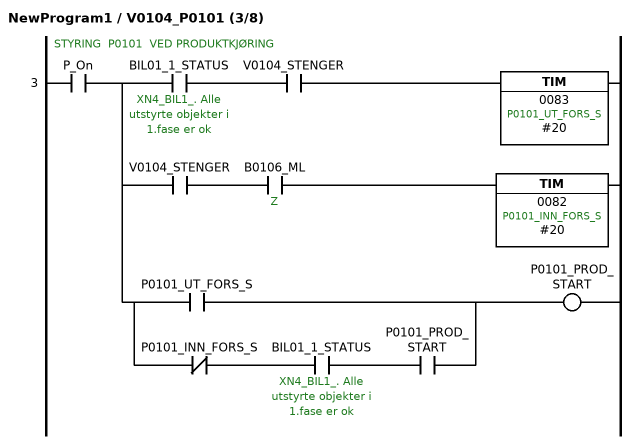
; rung 3: STYRING  P0101  VED PRODUKTKJØRING
LD P_On
OUT TR0
AND BIL01_1_STATUS  ; XN4_BIL1_. Alle utstyrte objekter i 1.fase er ok
AND V0104_STENGER
TIM 0083 #20  ; P0101_UT_FORS_S
LD TR0
AND V0104_STENGER
AND B0106_ML  ; Z
TIM 0082 #20  ; P0101_INN_FORS_S
LD TR0
LD P0101_UT_FORS_S
LDNOT P0101_INN_FORS_S
AND BIL01_1_STATUS  ; XN4_BIL1_. Alle utstyrte objekter i 1.fase er ok
AND P0101_PROD_START
ORLD
ANDLD
OUT P0101_PROD_START

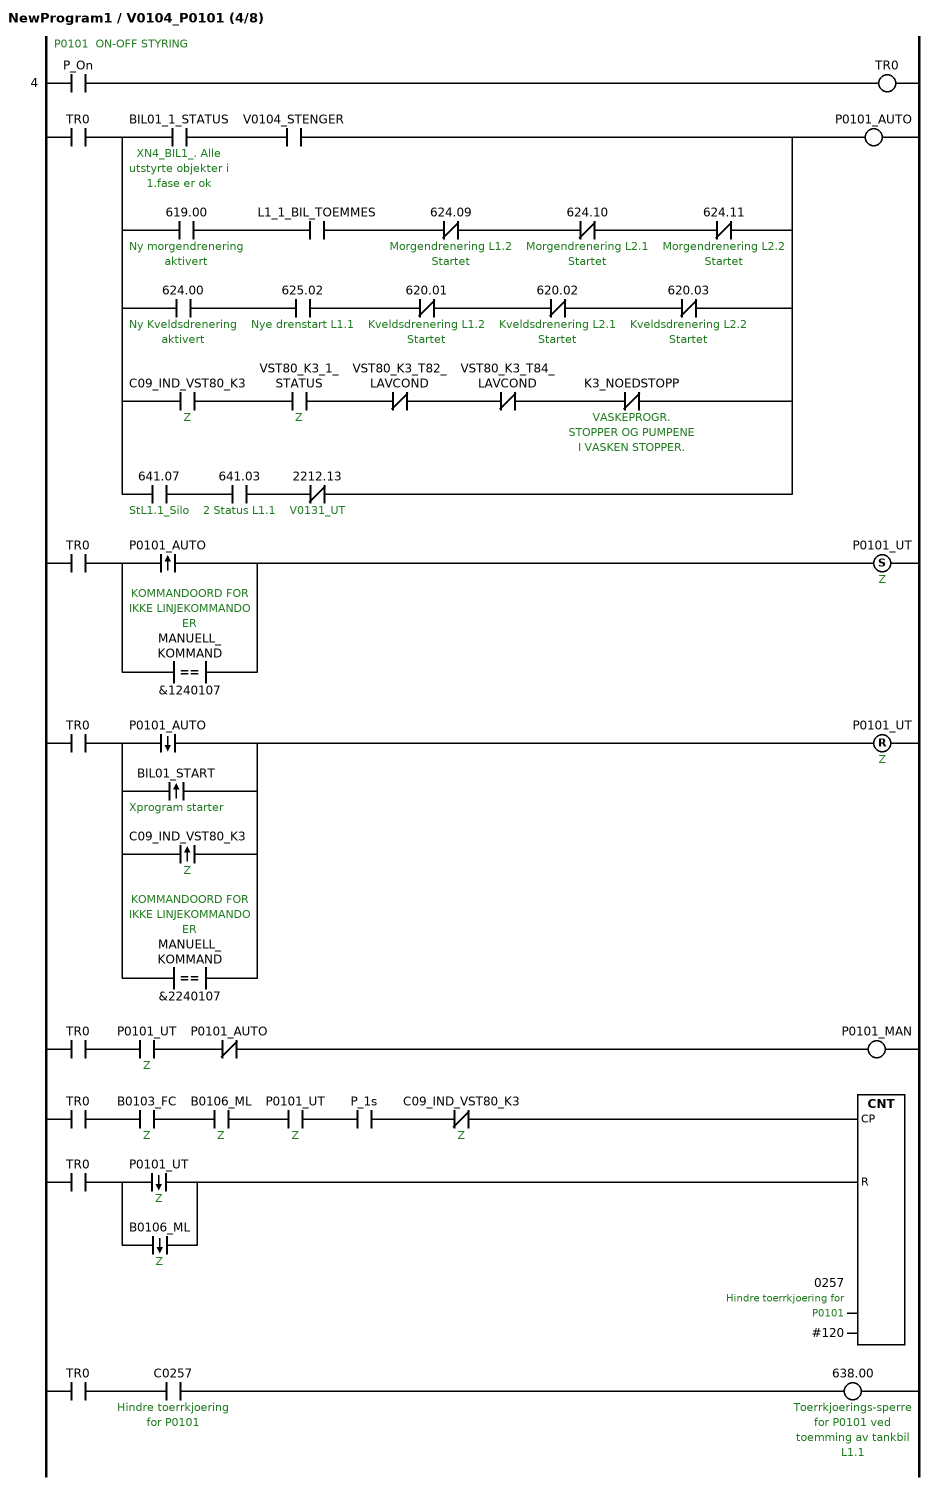
; rung 4: P0101  ON-OFF STYRING
LD P_On
OUT TR0
LD BIL01_1_STATUS  ; XN4_BIL1_. Alle utstyrte objekter i 1.fase er ok
AND V0104_STENGER
LD 619.00  ; Ny morgendrenering aktivert
AND L1_1_BIL_TOEMMES
ANDNOT 624.09  ; Morgendrenering L1.2 Startet
ANDNOT 624.10  ; Morgendrenering L2.1 Startet
ANDNOT 624.11  ; Morgendrenering L2.2 Startet
ORLD
LD 624.00  ; Ny Kveldsdrenering aktivert
AND 625.02  ; Nye drenstart L1.1
ANDNOT 620.01  ; Kveldsdrenering L1.2 Startet
ANDNOT 620.02  ; Kveldsdrenering L2.1 Startet
ANDNOT 620.03  ; Kveldsdrenering L2.2 Startet
ORLD
LD C09_IND_VST80_K3  ; Z
AND VST80_K3_1_STATUS  ; Z
ANDNOT VST80_K3_T82_LAVCOND
ANDNOT VST80_K3_T84_LAVCOND
ANDNOT K3_NOEDSTOPP  ; VASKEPROGR. STOPPER OG PUMPENE I VASKEN STOPPER.
ORLD
LD 641.07  ; StL1.1_Silo
AND 641.03  ; 2 Status L1.1
ANDNOT 2212.13  ; V0131_UT
ORLD
ANDLD
OUT P0101_AUTO
LD TR0
@LD P0101_AUTO
OR=L(301) MANUELL_KOMMAND &1240107  ; KOMMANDOORD FOR IKKE LINJEKOMMANDOER
ANDLD
SET P0101_UT  ; Z
LD TR0
%LD P0101_AUTO
@OR BIL01_START  ; Xprogram starter
@OR C09_IND_VST80_K3  ; Z
OR=L(301) MANUELL_KOMMAND &2240107  ; KOMMANDOORD FOR IKKE LINJEKOMMANDOER
ANDLD
RSET P0101_UT  ; Z
LD TR0
AND P0101_UT  ; Z
ANDNOT P0101_AUTO
OUT P0101_MAN
LD TR0
AND B0103_FC  ; Z
AND B0106_ML  ; Z
AND P0101_UT  ; Z
AND P_1s
ANDNOT C09_IND_VST80_K3  ; Z
LD TR0
%LD P0101_UT  ; Z
%OR B0106_ML  ; Z
ANDLD
CNT 0257 #120  ; Hindre toerrkjoering for P0101
LD TR0
AND C0257  ; Hindre toerrkjoering for P0101
OUT 638.00  ; Toerrkjoerings-sperre for P0101 ved toemming av tankbil L1.1

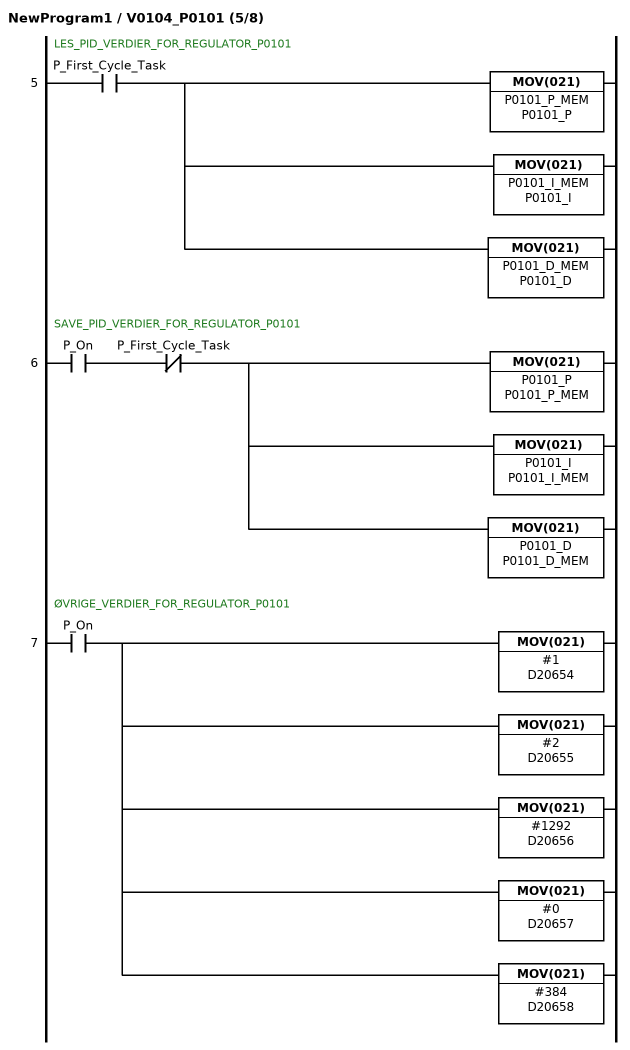
; rung 5: LES_PID_VERDIER_FOR_REGULATOR_P0101
LD P_First_Cycle_Task
MOV(021) P0101_P_MEM P0101_P
MOV(021) P0101_I_MEM P0101_I
MOV(021) P0101_D_MEM P0101_D
; rung 6: SAVE_PID_VERDIER_FOR_REGULATOR_P0101
LD P_On
ANDNOT P_First_Cycle_Task
MOV(021) P0101_P P0101_P_MEM
MOV(021) P0101_I P0101_I_MEM
MOV(021) P0101_D P0101_D_MEM
; rung 7: ØVRIGE_VERDIER_FOR_REGULATOR_P0101
LD P_On
MOV(021) #1 D20654
MOV(021) #2 D20655
MOV(021) #1292 D20656
MOV(021) #0 D20657
MOV(021) #384 D20658

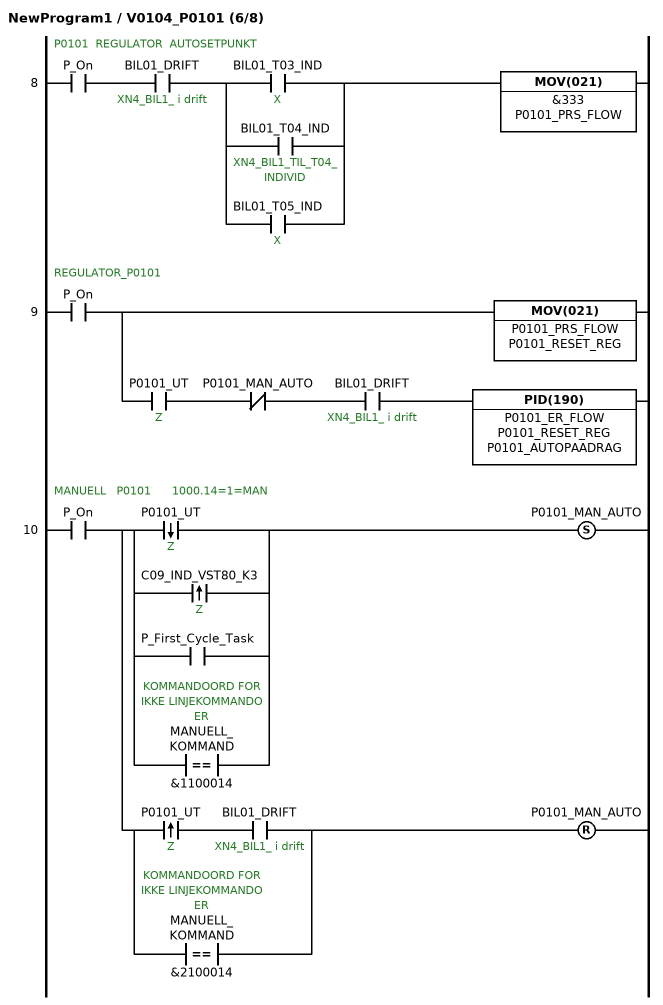
; rung 8: P0101  REGULATOR  AUTOSETPUNKT
LD P_On
AND BIL01_DRIFT  ; XN4_BIL1_ i drift
LD BIL01_T03_IND  ; X
OR BIL01_T04_IND  ; XN4_BIL1_TIL_T04_INDIVID
OR BIL01_T05_IND  ; X
ANDLD
MOV(021) &333 P0101_PRS_FLOW
; rung 9: REGULATOR_P0101
LD P_On
MOV(021) P0101_PRS_FLOW P0101_RESET_REG
AND P0101_UT  ; Z
ANDNOT P0101_MAN_AUTO
AND BIL01_DRIFT  ; XN4_BIL1_ i drift
PID(190) P0101_ER_FLOW P0101_RESET_REG P0101_AUTOPAADRAG
; rung 10: MANUELL   P0101      1000.14=1=MAN
LD P_On
OUT TR0
%LD P0101_UT  ; Z
@OR C09_IND_VST80_K3  ; Z
OR P_First_Cycle_Task
OR=L(301) MANUELL_KOMMAND &1100014  ; KOMMANDOORD FOR IKKE LINJEKOMMANDOER
ANDLD
SET P0101_MAN_AUTO
LD TR0
@LD P0101_UT  ; Z
AND BIL01_DRIFT  ; XN4_BIL1_ i drift
OR=L(301) MANUELL_KOMMAND &2100014  ; KOMMANDOORD FOR IKKE LINJEKOMMANDOER
ANDLD
RSET P0101_MAN_AUTO

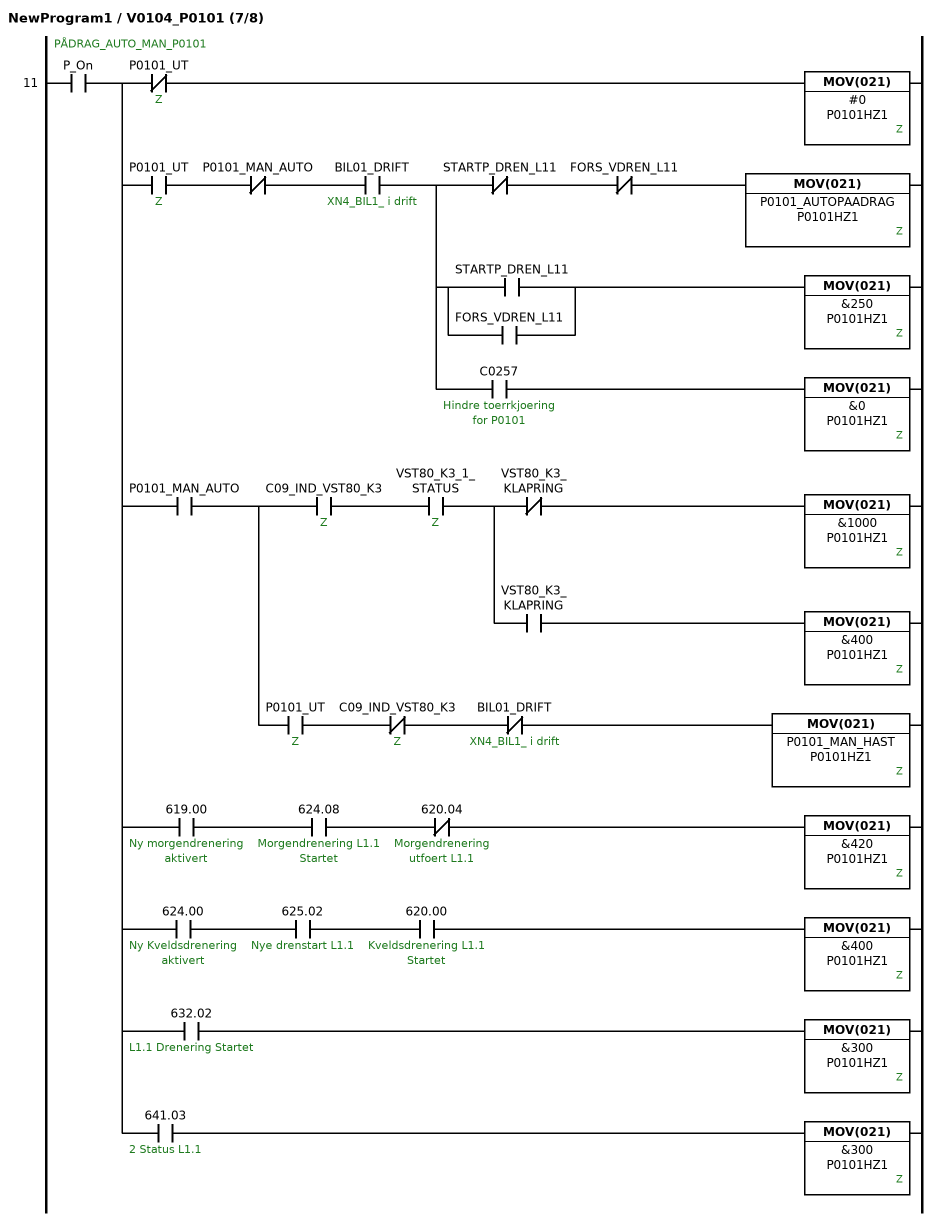
; rung 11: PÅDRAG_AUTO_MAN_P0101
LD P_On
OUT TR0
ANDNOT P0101_UT  ; Z
MOV(021) #0 P0101HZ1  ; Z
LD TR0
AND P0101_UT  ; Z
ANDNOT P0101_MAN_AUTO
AND BIL01_DRIFT  ; XN4_BIL1_ i drift
OUT TR1
ANDNOT STARTP_DREN_L11
ANDNOT FORS_VDREN_L11
MOV(021) P0101_AUTOPAADRAG P0101HZ1  ; Z
LD TR1
LD STARTP_DREN_L11
OR FORS_VDREN_L11
ANDLD
MOV(021) &250 P0101HZ1  ; Z
LD TR1
AND C0257  ; Hindre toerrkjoering for P0101
MOV(021) &0 P0101HZ1  ; Z
LD TR0
AND P0101_MAN_AUTO
OUT TR1
AND C09_IND_VST80_K3  ; Z
AND VST80_K3_1_STATUS  ; Z
OUT TR2
ANDNOT VST80_K3_KLAPRING
MOV(021) &1000 P0101HZ1  ; Z
LD TR2
AND VST80_K3_KLAPRING
MOV(021) &400 P0101HZ1  ; Z
LD TR1
AND P0101_UT  ; Z
ANDNOT C09_IND_VST80_K3  ; Z
ANDNOT BIL01_DRIFT  ; XN4_BIL1_ i drift
MOV(021) P0101_MAN_HAST P0101HZ1  ; Z
LD TR0
AND 619.00  ; Ny morgendrenering aktivert
AND 624.08  ; Morgendrenering L1.1 Startet
ANDNOT 620.04  ; Morgendrenering utfoert L1.1
MOV(021) &420 P0101HZ1  ; Z
LD TR0
AND 624.00  ; Ny Kveldsdrenering aktivert
AND 625.02  ; Nye drenstart L1.1
AND 620.00  ; Kveldsdrenering L1.1 Startet
MOV(021) &400 P0101HZ1  ; Z
LD TR0
AND 632.02  ; L1.1 Drenering Startet
MOV(021) &300 P0101HZ1  ; Z
LD TR0
AND 641.03  ; 2 Status L1.1
MOV(021) &300 P0101HZ1  ; Z

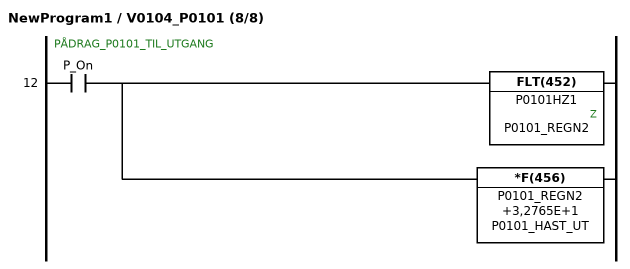
; rung 12: PÅDRAG_P0101_TIL_UTGANG
LD P_On
FLT(452) P0101HZ1 P0101_REGN2  ; Z
*F(456) P0101_REGN2 +3,2765E+1 P0101_HAST_UT
; rung 13: Ingen_kommentar_funnet

### Section P0102_ISVANN

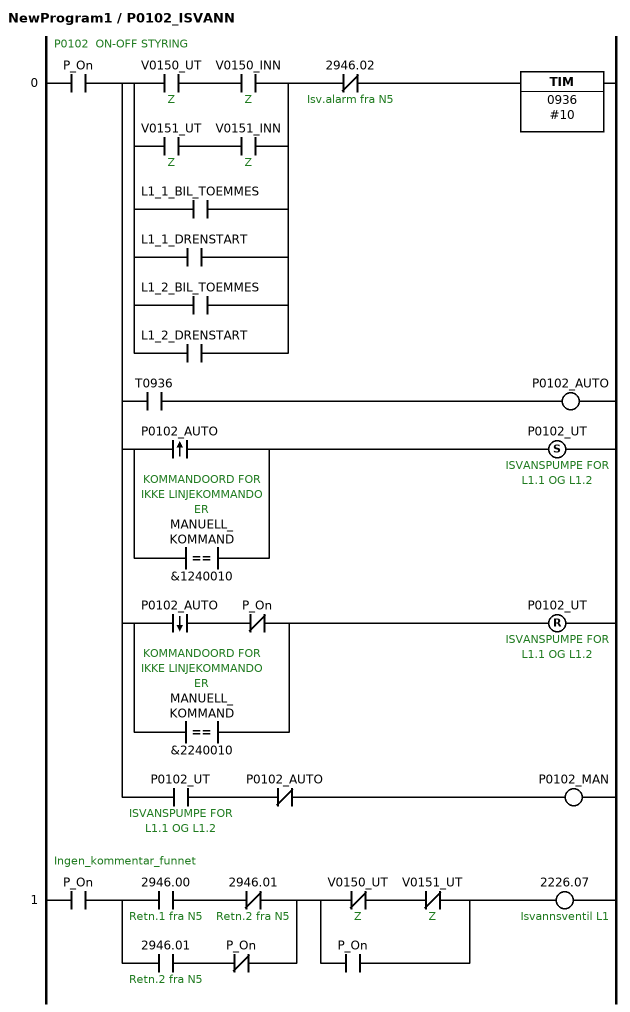
; rung 0: P0102  ON-OFF STYRING
LD P_On
OUT TR0
LD V0150_UT  ; Z
AND V0150_INN  ; Z
LD V0151_UT  ; Z
AND V0151_INN  ; Z
ORLD
OR L1_1_BIL_TOEMMES
OR L1_1_DRENSTART
OR L1_2_BIL_TOEMMES
OR L1_2_DRENSTART
ANDLD
ANDNOT 2946.02  ; Isv.alarm fra N5
TIM 0936 #10
LD TR0
AND T0936
OUT P0102_AUTO
LD TR0
@LD P0102_AUTO
OR=L(301) MANUELL_KOMMAND &1240010  ; KOMMANDOORD FOR IKKE LINJEKOMMANDOER
ANDLD
SET P0102_UT  ; ISVANSPUMPE FOR L1.1 OG L1.2
LD TR0
%LD P0102_AUTO
ANDNOT P_On
OR=L(301) MANUELL_KOMMAND &2240010  ; KOMMANDOORD FOR IKKE LINJEKOMMANDOER
ANDLD
RSET P0102_UT  ; ISVANSPUMPE FOR L1.1 OG L1.2
LD TR0
AND P0102_UT  ; ISVANSPUMPE FOR L1.1 OG L1.2
ANDNOT P0102_AUTO
OUT P0102_MAN
; rung 1: Ingen_kommentar_funnet
LD P_On
LD 2946.00  ; Retn.1 fra N5
ANDNOT 2946.01  ; Retn.2 fra N5
LD 2946.01  ; Retn.2 fra N5
ANDNOT P_On
ORLD
ANDLD
LDNOT V0150_UT  ; Z
ANDNOT V0151_UT  ; Z
OR P_On
ANDLD
OUT 2226.07  ; Isvannsventil L1
; rung 2: Ingen_kommentar_funnet

### Section V0150_V0153_ISV

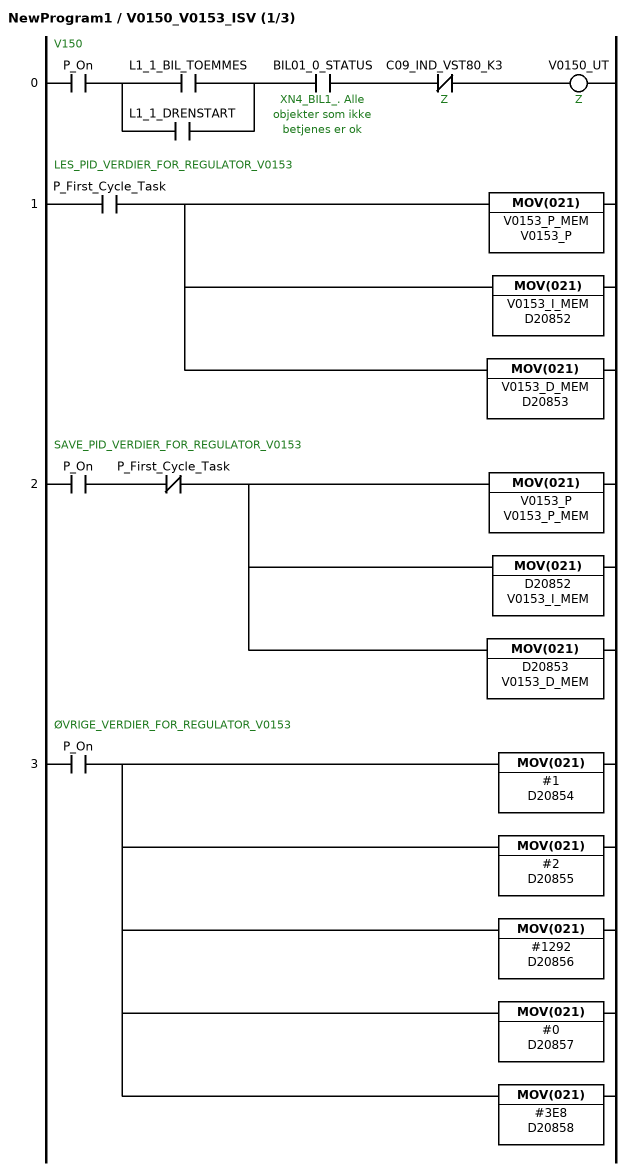
; rung 0: V150
LD P_On
LD L1_1_BIL_TOEMMES
OR L1_1_DRENSTART
ANDLD
AND BIL01_0_STATUS  ; XN4_BIL1_. Alle objekter som ikke betjenes er ok
ANDNOT C09_IND_VST80_K3  ; Z
OUT V0150_UT  ; Z
; rung 1: LES_PID_VERDIER_FOR_REGULATOR_V0153
LD P_First_Cycle_Task
MOV(021) V0153_P_MEM V0153_P
MOV(021) V0153_I_MEM D20852
MOV(021) V0153_D_MEM D20853
; rung 2: SAVE_PID_VERDIER_FOR_REGULATOR_V0153
LD P_On
ANDNOT P_First_Cycle_Task
MOV(021) V0153_P V0153_P_MEM
MOV(021) D20852 V0153_I_MEM
MOV(021) D20853 V0153_D_MEM
; rung 3: ØVRIGE_VERDIER_FOR_REGULATOR_V0153
LD P_On
MOV(021) #1 D20854
MOV(021) #2 D20855
MOV(021) #1292 D20856
MOV(021) #0 D20857
MOV(021) #3E8 D20858

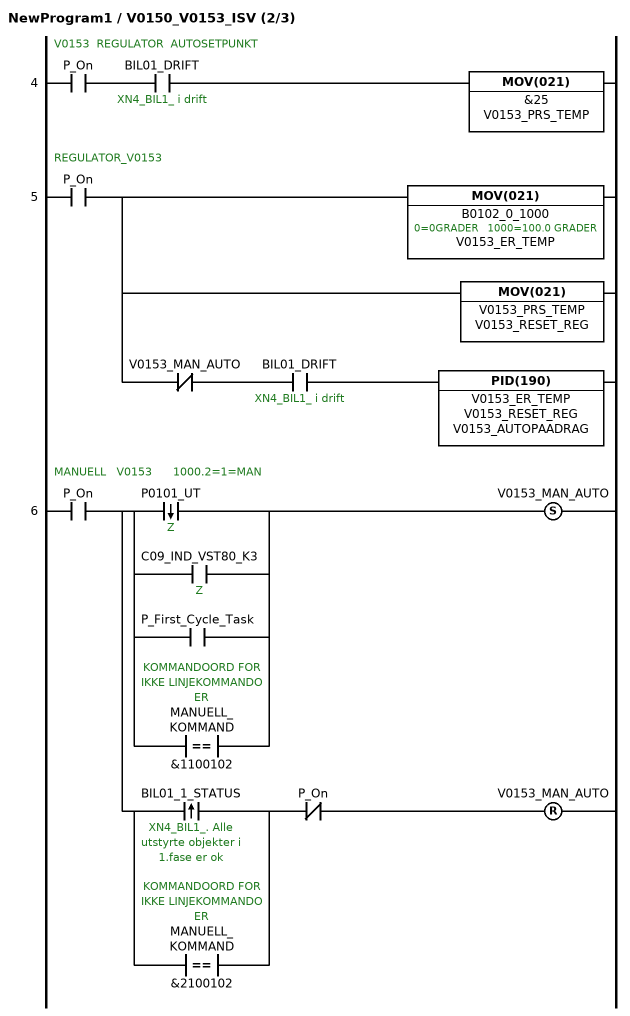
; rung 4: V0153  REGULATOR  AUTOSETPUNKT
LD P_On
AND BIL01_DRIFT  ; XN4_BIL1_ i drift
MOV(021) &25 V0153_PRS_TEMP
; rung 5: REGULATOR_V0153
LD P_On
MOV(021) B0102_0_1000 V0153_ER_TEMP  ; 0=0GRADER   1000=100.0 GRADER
MOV(021) V0153_PRS_TEMP V0153_RESET_REG
ANDNOT V0153_MAN_AUTO
AND BIL01_DRIFT  ; XN4_BIL1_ i drift
PID(190) V0153_ER_TEMP V0153_RESET_REG V0153_AUTOPAADRAG
; rung 6: MANUELL   V0153      1000.2=1=MAN
LD P_On
OUT TR0
%LD P0101_UT  ; Z
OR C09_IND_VST80_K3  ; Z
OR P_First_Cycle_Task
OR=L(301) MANUELL_KOMMAND &1100102  ; KOMMANDOORD FOR IKKE LINJEKOMMANDOER
ANDLD
SET V0153_MAN_AUTO
LD TR0
@LD BIL01_1_STATUS  ; XN4_BIL1_. Alle utstyrte objekter i 1.fase er ok
OR=L(301) MANUELL_KOMMAND &2100102  ; KOMMANDOORD FOR IKKE LINJEKOMMANDOER
ANDLD
ANDNOT P_On
RSET V0153_MAN_AUTO

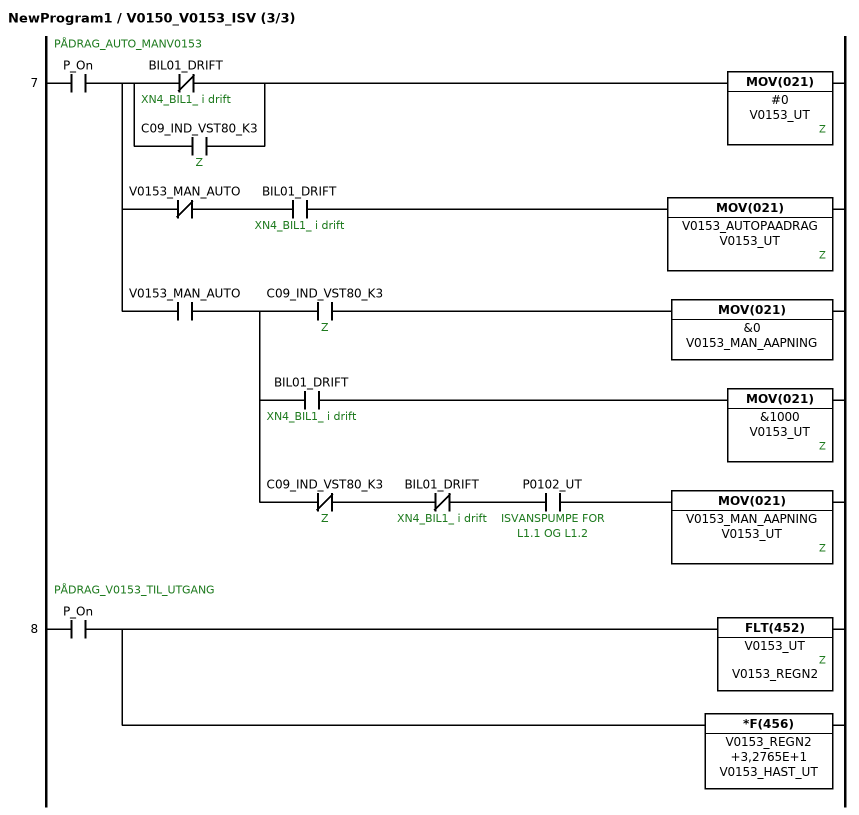
; rung 7: PÅDRAG_AUTO_MANV0153
LD P_On
OUT TR0
LDNOT BIL01_DRIFT  ; XN4_BIL1_ i drift
OR C09_IND_VST80_K3  ; Z
ANDLD
MOV(021) #0 V0153_UT  ; Z
LD TR0
ANDNOT V0153_MAN_AUTO
AND BIL01_DRIFT  ; XN4_BIL1_ i drift
MOV(021) V0153_AUTOPAADRAG V0153_UT  ; Z
LD TR0
AND V0153_MAN_AUTO
OUT TR0
AND C09_IND_VST80_K3  ; Z
MOV(021) &0 V0153_MAN_AAPNING
LD TR0
AND BIL01_DRIFT  ; XN4_BIL1_ i drift
MOV(021) &1000 V0153_UT  ; Z
LD TR0
ANDNOT C09_IND_VST80_K3  ; Z
ANDNOT BIL01_DRIFT  ; XN4_BIL1_ i drift
AND P0102_UT  ; ISVANSPUMPE FOR L1.1 OG L1.2
MOV(021) V0153_MAN_AAPNING V0153_UT  ; Z
; rung 8: PÅDRAG_V0153_TIL_UTGANG
LD P_On
FLT(452) V0153_UT V0153_REGN2  ; Z
*F(456) V0153_REGN2 +3,2765E+1 V0153_HAST_UT
; rung 9: Ingen_kommentar_funnet

### Section PGM_521_HENGER01_L1_2_TIL_SILO

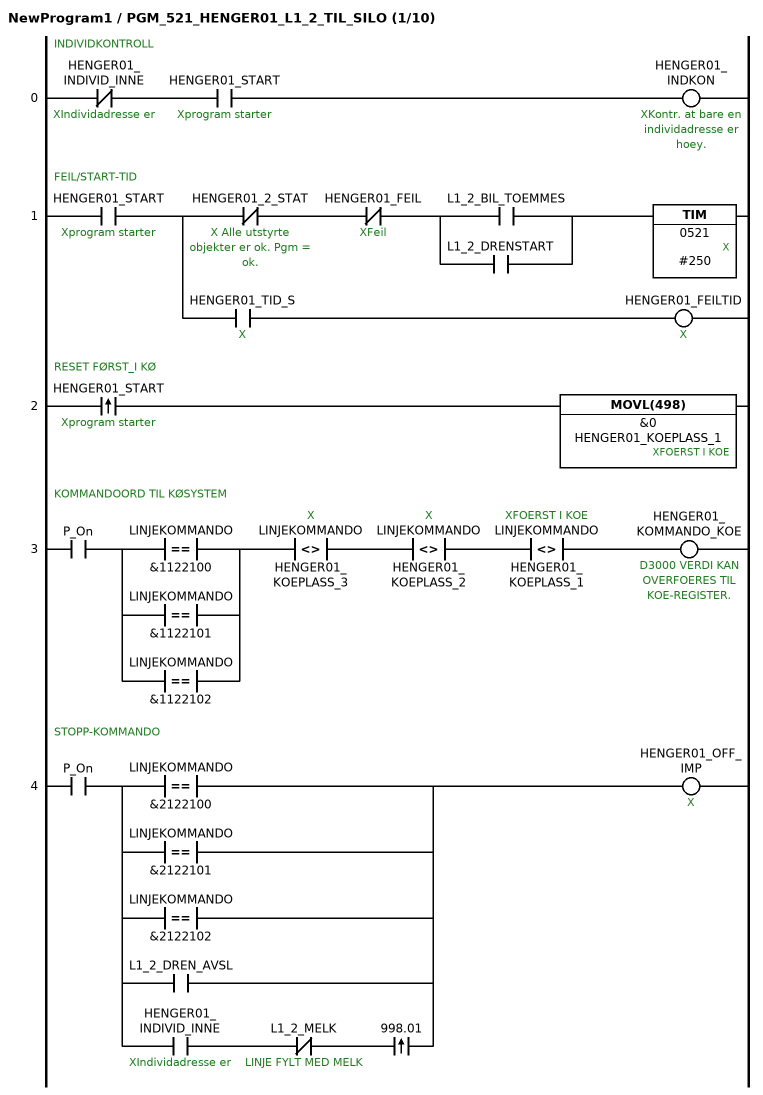
; rung 0: INDIVIDKONTROLL
LDNOT HENGER01_INDIVID_INNE  ; XIndividadresse er
AND HENGER01_START  ; Xprogram starter
OUT HENGER01_INDKON  ; XKontr. at bare en individadresse er hoey.
; rung 1: FEIL/START-TID
LD HENGER01_START  ; Xprogram starter
OUT TR0
ANDNOT HENGER01_2_STAT  ; X Alle utstyrte objekter er ok. Pgm = ok.
ANDNOT HENGER01_FEIL  ; XFeil
LD L1_2_BIL_TOEMMES
OR L1_2_DRENSTART
ANDLD
TIM 0521 #250  ; X
LD TR0
AND HENGER01_TID_S  ; X
OUT HENGER01_FEILTID  ; X
; rung 2: RESET FØRST_I KØ
@LD HENGER01_START  ; Xprogram starter
MOVL(498) &0 HENGER01_KOEPLASS_1  ; XFOERST I KOE
; rung 3: KOMMANDOORD TIL KØSYSTEM
LD P_On
LD=L(301) LINJEKOMMANDO &1122100
OR=L(301) LINJEKOMMANDO &1122101
OR=L(301) LINJEKOMMANDO &1122102
ANDLD
AND<>L(306) LINJEKOMMANDO HENGER01_KOEPLASS_3  ; X
AND<>L(306) LINJEKOMMANDO HENGER01_KOEPLASS_2  ; X
AND<>L(306) LINJEKOMMANDO HENGER01_KOEPLASS_1  ; XFOERST I KOE
OUT HENGER01_KOMMANDO_KOE  ; D3000 VERDI KAN OVERFOERES TIL KOE-REGISTER.
; rung 4: STOPP-KOMMANDO
LD P_On
LD=L(301) LINJEKOMMANDO &2122100
OR=L(301) LINJEKOMMANDO &2122101
OR=L(301) LINJEKOMMANDO &2122102
OR L1_2_DREN_AVSL
LD HENGER01_INDIVID_INNE  ; XIndividadresse er
ANDNOT L1_2_MELK  ; LINJE FYLT MED MELK
@AND 998.01
ORLD
ANDLD
OUT HENGER01_OFF_IMP  ; X

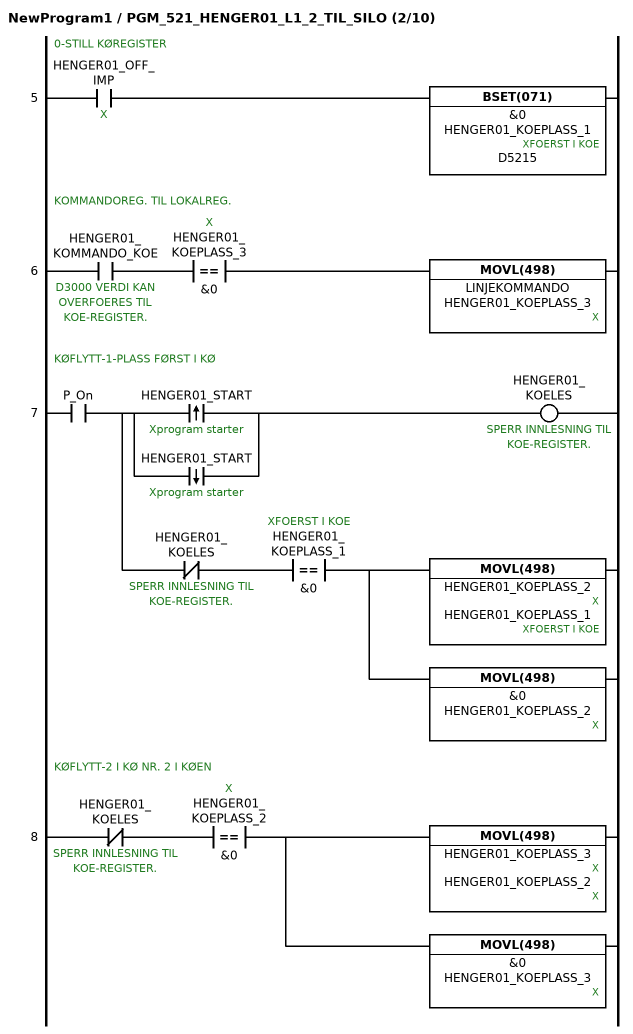
; rung 5: 0-STILL KØREGISTER
LD HENGER01_OFF_IMP  ; X
BSET(071) &0 HENGER01_KOEPLASS_1 D5215  ; XFOERST I KOE
; rung 6: KOMMANDOREG. TIL LOKALREG.
LD HENGER01_KOMMANDO_KOE  ; D3000 VERDI KAN OVERFOERES TIL KOE-REGISTER.
AND=L(301) HENGER01_KOEPLASS_3 &0  ; X
MOVL(498) LINJEKOMMANDO HENGER01_KOEPLASS_3  ; X
; rung 7: KØFLYTT-1-PLASS FØRST I KØ
LD P_On
OUT TR0
@LD HENGER01_START  ; Xprogram starter
%OR HENGER01_START  ; Xprogram starter
ANDLD
OUT HENGER01_KOELES  ; SPERR INNLESNING TIL KOE-REGISTER.
LD TR0
ANDNOT HENGER01_KOELES  ; SPERR INNLESNING TIL KOE-REGISTER.
AND=L(301) HENGER01_KOEPLASS_1 &0  ; XFOERST I KOE
MOVL(498) HENGER01_KOEPLASS_2 HENGER01_KOEPLASS_1  ; X, XFOERST I KOE
MOVL(498) &0 HENGER01_KOEPLASS_2  ; X
; rung 8: KØFLYTT-2 I KØ NR. 2 I KØEN
LDNOT HENGER01_KOELES  ; SPERR INNLESNING TIL KOE-REGISTER.
AND=L(301) HENGER01_KOEPLASS_2 &0  ; X
MOVL(498) HENGER01_KOEPLASS_3 HENGER01_KOEPLASS_2  ; X
MOVL(498) &0 HENGER01_KOEPLASS_3  ; X

